PROGRAM AXES_CYCLE
VAR
END_VAR

GRP1();

ACTION GRP1:
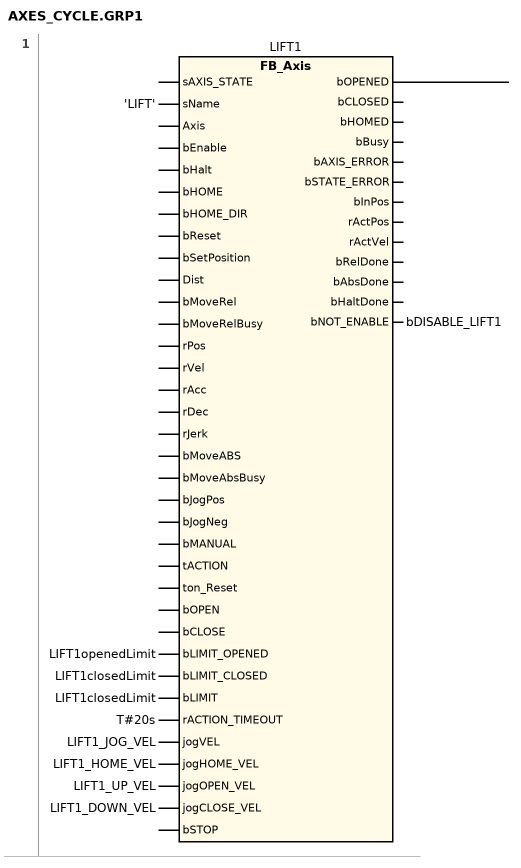
// NETWORK 1
LIFT1(
    sName := 'LIFT',
    bLIMIT_OPENED := LIFT1openedLimit,
    bLIMIT_CLOSED := LIFT1closedLimit,
    bLIMIT := LIFT1closedLimit,
    rACTION_TIMEOUT := T#20s,
    jogVEL := LIFT1_JOG_VEL,
    jogHOME_VEL := LIFT1_HOME_VEL,
    jogOPEN_VEL := LIFT1_UP_VEL,
    jogCLOSE_VEL := LIFT1_DOWN_VEL,
    bNOT_ENABLE => bDISABLE_LIFT1); // FB_Axis

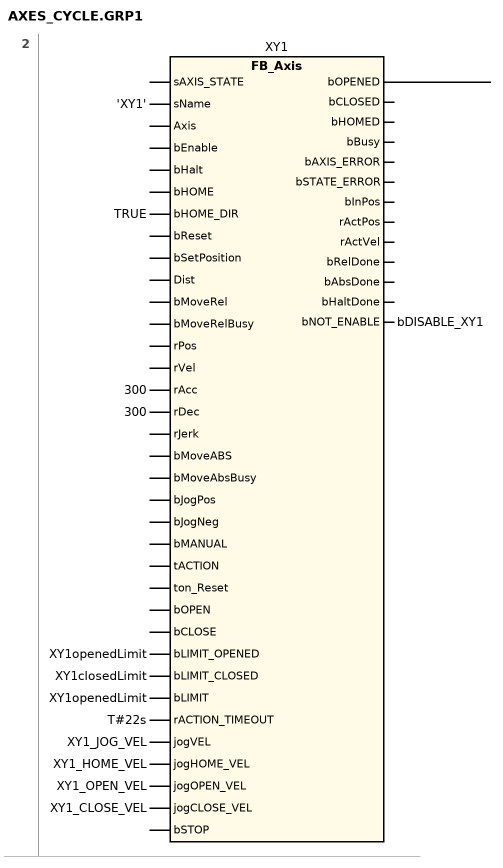
// NETWORK 2
XY1(
    sName := 'XY1',
    bHOME_DIR := TRUE,
    rAcc := 300,
    rDec := 300,
    bLIMIT_OPENED := XY1openedLimit,
    bLIMIT_CLOSED := XY1closedLimit,
    bLIMIT := XY1openedLimit,
    rACTION_TIMEOUT := T#22s,
    jogVEL := XY1_JOG_VEL,
    jogHOME_VEL := XY1_HOME_VEL,
    jogOPEN_VEL := XY1_OPEN_VEL,
    jogCLOSE_VEL := XY1_CLOSE_VEL,
    bNOT_ENABLE => bDISABLE_XY1); // FB_Axis

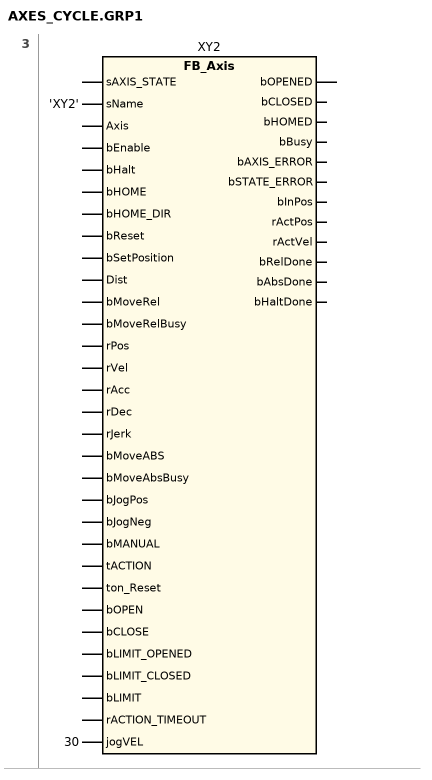
// NETWORK 3
XY2(sName := 'XY2', jogVEL := 30); // FB_Axis

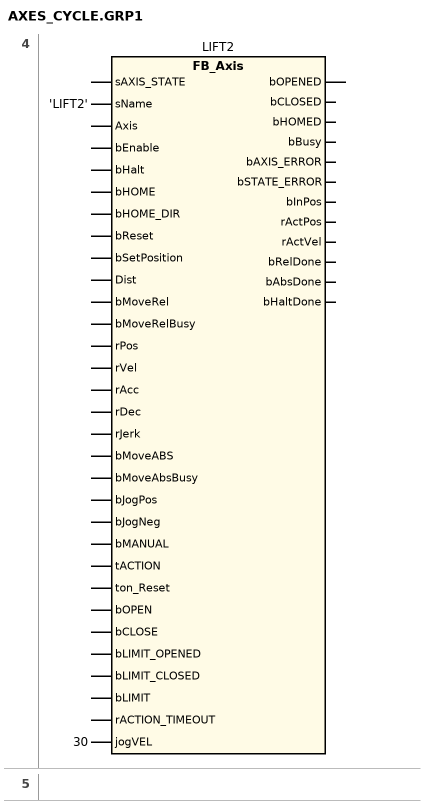
// NETWORK 4
LIFT2(sName := 'LIFT2', jogVEL := 30); // FB_Axis

// NETWORK 5
END_ACTION

END_PROGRAM

(* stored: Version 1.1.0.1, ProductVersion 3.1.4024.12
   POU AXES_CYCLE: Id {9cd0cba8-0116-4d06-bcad-bfddb259f9ba}, SpecialFunc None
   Action GRP1: Id {c92a8f88-fc9a-4b1d-835c-ccf46ea4c98c} *)
